Fanuc KAREL source: kt00122.KL

-- PROVISIONAL review KL for V770-1; original PC SHA256 573886de19e9aef23eec37356068987b4e1ab23f7ee3f7846eb8f59e65a776b3
-- Incomplete behavior may be omitted. Consult companion uncertainty JSON. Do not deploy.
PROGRAM KT00122
%NOLOCKGROUP
VAR
  I2 : INTEGER
  OUT : REAL
-- UNRESOLVED_DECL H1 type=002017
BEGIN
  -- UNRESOLVED_PC offsets 5-19; opcodes 2E,22,9D,33,B4
  -- UNRESOLVED_PC offsets 24-35; opcodes 2E,23
  -- UNRESOLVED_PC offsets 40-66; opcodes 22,9D,33,B3,21,64,29,64,29,6C,23
  -- UNRESOLVED_PC offsets 71-75; opcodes 7F
END KT00122
